(* CoDeSys 2.3.9.37 project: Cap9_1_Res.pro *)
(* Libraries: Standard.LIB 4.10.05 12:14:46 *)

(* Global variable list: Global_Variables *)
VAR_GLOBAL

(* Variables de entrada *)
    Numero: INT ;


(* Variables de Salida*)
      a0:BOOL;
	b0:BOOL;
	c0:BOOL;
	d0:BOOL;
	e0:BOOL;
	f0:BOOL;
	g0:BOOL;
      Novalido:BOOL;

END_VAR

(* POU PLC_PRG, ST *)
PROGRAM PLC_PRG
VAR
 MiDisplay: SieteSegmentos;
END_VAR
MiDisplay(Digito:=Numero,a=>a0,b=>b0,
                  c=>c0,d=>d0,e=>e0,f=>f0,g=>g0);
Novalido:=MiDisplay.Error;
END_PROGRAM

(* POU SieteSegmentos, ST *)
FUNCTION_BLOCK SieteSegmentos
VAR_INPUT
    Digito:INT;
END_VAR
VAR_OUTPUT
    a :BOOL;
   b :BOOL;
   c :BOOL;
   d :BOOL;
   e :BOOL;
   f :BOOL;
   g :BOOL;
  Error :BOOL;
END_VAR
VAR
END_VAR
 Error:=Digito<0 OR Digito>9;
   a:=FALSE;  b:=FALSE;  c:=FALSE;  d:=FALSE;
   e:=FALSE; f:=FALSE; g:=FALSE;
IF NOT Error THEN
   CASE Digito OF
      0:  a:=TRUE; b:=TRUE; c:=TRUE; d:=TRUE; e:=TRUE; f:=TRUE;
      1: b:=TRUE; c:=TRUE;
      2: a:=TRUE; b:=TRUE; g:=TRUE; e:=TRUE; d:=TRUE;
      3: a:=TRUE; b:=TRUE; c:=TRUE; d:=TRUE; g:=TRUE;
      4: b:=TRUE; g:=TRUE;f:=TRUE;c:=TRUE;
      5: a:=TRUE;c:=TRUE;d:=TRUE;f:=TRUE;g:=TRUE;
	6:a:=TRUE; c:=TRUE; d:=TRUE; e:=TRUE; f:=TRUE;g:=TRUE;
      8: a:=TRUE; b:=TRUE; c:=TRUE; d:=TRUE; e:=TRUE; f:=TRUE;g:=TRUE;
      7:a:=TRUE;b:=TRUE;c:=TRUE;
      9:a:=TRUE; b:=TRUE; c:=TRUE; d:=TRUE; f:=TRUE;g:=TRUE;
    END_CASE;


  END_IF
END_FUNCTION_BLOCK

(* Visualisation Display
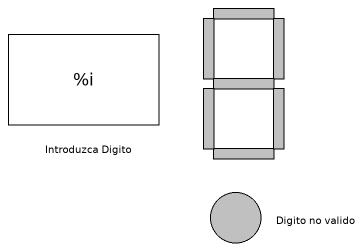
rectangle at (265,64)-(326,75): alarm colour if a0
rectangle at (325,74)-(336,135): alarm colour if b0
rectangle at (255,74)-(266,135): alarm colour if f0
rectangle at (265,134)-(326,145): alarm colour if g0
rectangle at (265,204)-(326,215): alarm colour if d0
rectangle at (325,144)-(336,205): alarm colour if c0
rectangle at (255,144)-(266,205): alarm colour if e0
rectangle at (60,90)-(211,181): text "%i"; shows Numero; editable
ellipse at (262,248)-(313,299): alarm colour if Novalido
rectangle at (60,190)-(221,221): text "Introduzca Digito"
rectangle at (287,261)-(448,292): text "Digito no valido"
*)
